FUNCTION_BLOCK OnStackDisposedHandler EXTENDS OnStackEventHandler

METHOD PUBLIC HandleEvent
VAR_INPUT
	Event : I_Event;
END_VAR
VAR
	stackDisposedEvent : I_StackDisposedEvent;
END_VAR
IF __QUERYINTERFACE(Event, stackDisposedEvent) THEN
	_eventReceived := TRUE;
	fromExpected := stackDisposedEvent.TargetStack = expectedOriginator;
END_IF
END_METHOD

END_FUNCTION_BLOCK

(* stored: Version 1.1.0.1, ProductVersion 3.1.4024.12
   POU OnStackDisposedHandler: Id {587df8cf-8687-4c59-bb92-5dd1ae2c7f81}, SpecialFunc None
   Method HandleEvent: Id {59c23e56-56fb-4891-be13-7116b741a739} *)
